(* PLC project Unnamed, Unknown Unnamed 1 *)
(* stored: creationDateTime 2013-01-29T14:01:00, modificationDateTime 2013-02-26T15:59:13 *)

FUNCTION_BLOCK WORD_AS_REAL
  VAR_OUTPUT
    out : REAL;
  END_VAR
  VAR_INPUT
    inHigh : WORD;
    inLow : WORD;
  END_VAR

                        OUT := 0.0;
                        {{
                        	unsigned int *p =(unsigned int*)&GetFbVar(OUT);
                            *p = (unsigned short int)GetFbVar(INLOW);
                            *p |= ((unsigned short int)GetFbVar(INHIGH))<<16;
                        ;}}
                    
END_FUNCTION_BLOCK

FUNCTION_BLOCK REAL_AS_WORD
  VAR_INPUT
    in : REAL;
  END_VAR
  VAR_OUTPUT
    outHigh : WORD;
    outLow : WORD;
  END_VAR

                        outHigh := INT_TO_WORD(0);
                        outLow := INT_TO_WORD(0);
                        {{
                            unsigned int *src = (unsigned int*) &GetFbVar(IN);
                            GetFbVar(OUTHIGH) = ((*src)>>16) & 0xFFFF;
                            GetFbVar(OUTLOW) = *src & 0xFFFF;
                        ;}}
                    
END_FUNCTION_BLOCK
